{attribute addProperty BoxType "EPP2316-0003-0016"}
{attribute addProperty Id "Set_safe_stateAT %Q*BOOL811Reset_outputsAT %Q*BOOL812"}
{attribute addProperty CRC "1934623490"}
{attribute addProperty SizeInBites "16"}
{attribute addProperty SizeInBytes "2"}
TYPE DIG_Outputs_Device_73500302 :
STRUCT
	{attribute addProperty Name "Set_safe_state"}
	Set_safe_state AT %Q* : BOOL;
	{attribute addProperty Name "Reset_outputs"}
	Reset_outputs AT %Q* : BOOL;
END_STRUCT
END_TYPE

(* stored: Version 1.2.0.0, ProductVersion 3.1.4024.9
   DUT DIG_Outputs_Device_73500302: Id {7621a27d-5a77-4b76-aa3e-991057a9bacd} *)
